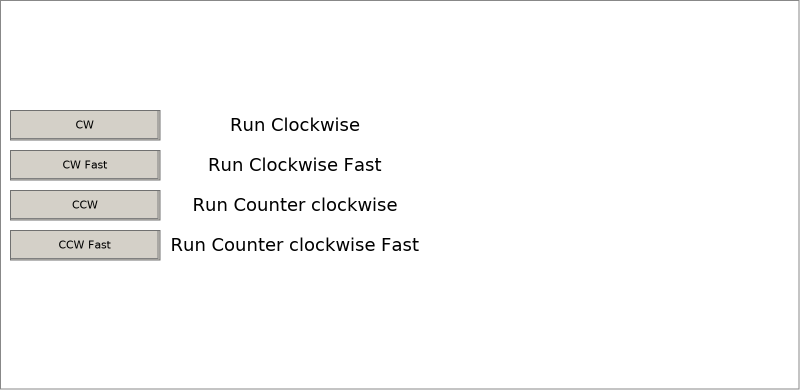
VISUALIZATION VisuTwoVelocityAxisControl  // 800x390
VAR_IN_OUT
	fbManualControler	: FB_ManualController ;
END_VAR
    Button (10,110 150x30), "CW"
        tap fbManualControler.pDevTwoVelocityAxis^.stManualControl.bManRunCW
    Button (10,150 150x30), "CW Fast"
        tap fbManualControler.pDevTwoVelocityAxis^.stManualControl.bManRunCWFast
    Button (10,190 150x30), "CCW"
        tap fbManualControler.pDevTwoVelocityAxis^.stManualControl.bManRunCCw
    Button (10,230 150x30), "CCW Fast"
        tap fbManualControler.pDevTwoVelocityAxis^.stManualControl.bManRunCCWFast
    Label (170,110 250x30), "Run Clockwise"
    Label (170,150 250x30), "Run Clockwise Fast"
    Label (170,190 250x30), "Run Counter clockwise"
    Label (170,230 250x30), "Run Counter clockwise Fast"
END_VISUALIZATION

(* stored: Version 1.1.0.1, ProductVersion 3.1.4024.10
   Visu VisuTwoVelocityAxisControl: Id {f7ef9a45-5a40-4a4e-8911-e78982b2c15b} *)
